// TIA Portal V17 export
// export: Created 2026-07-07T17:35:54.3389867Z, ExportSetting WithDefaults, DisplayName Totally Integrated Automation Portal, DisplayVersion V17, DisplayName TIA Portal Openness, DisplayVersion V17, DisplayName TIA Portal Version Control Interface, DisplayVersion V17, DisplayName STEP 7 Professional, DisplayVersion V17, DisplayName STEP 7 Safety, DisplayVersion V17, DisplayName WinCC Professional, DisplayVersion V17
FUNCTION_BLOCK "RS485_Com_Motor"   // FB2, LAD
TITLE = Feetech Motor with Cannet
{ S7_Optimized_Access := 'TRUE' }
VERSION : 0.1
// Note: Tcon block is required seperately for establishing the commincation.
// 
// Inputs:
// Connection_Done - Connection established bit from TCON block
// Slave_ID                  - Modbus RTU slave ID
// Target_Pos              - Input the Target position in Degrees
// Move                        - After giving the Target position this bit need to be enabled for executing. 
// 
// Outputs: 
// Actual_pos              - Gives the actual position in Degrees
// Target_Reached     - The bit will be enable for 2 seconds after the motor reaches the target position.
// stored: AutoNumber true, IsIECCheckEnabled false, IsRetainMemResEnabled false, MemoryReserve 100, SetENOAutomatically false, UDAEnableTagReadback false
   VAR_INPUT
      Connection_Done : Bool;
      Slave_ID : Int;
      Target_Pos : Int;
      Move : Bool;
   END_VAR
   VAR_OUTPUT
      "Actual_pos(Deg)" : Int;
      Target_Reached : Bool;
   END_VAR
   VAR
      CRC : Word;
      Frame_length : Int;
      CRC_Low : Byte;
      CRC_High : Byte;
      i : Int;
      j : Int;
      Data_Read { ExternalAccessible := 'False'; ExternalVisible := 'False'; ExternalWritable := 'False'} : Array[0..6] of Byte;
      Data_Write { ExternalAccessible := 'False'; ExternalVisible := 'False'; ExternalWritable := 'False'} : Array[0..7] of Byte;
      T_Send_block { S7_SetPoint := 'True'} : TSEND;
      T_RCV_Block { S7_SetPoint := 'True'} : TRCV;
      Move_timer { S7_SetPoint := 'True'} : IEC_TIMER;
      Send_req { S7_SetPoint := 'True'} : Bool;
      Function_code : Byte;
      Addr_low : Byte;
      Addr_high : Byte;
      Data_low : Byte;
      Data_high : Byte;
      Data_word : Word;
      Actual_pos_word : Word;
      Target_reach_timer : IEC_TIMER;
      Upper_limit { S7_SetPoint := 'True'} : Int;
      Lower_limit { S7_SetPoint := 'True'} : Int;
   END_VAR
BEGIN

REGION Network 1: Data send and recive
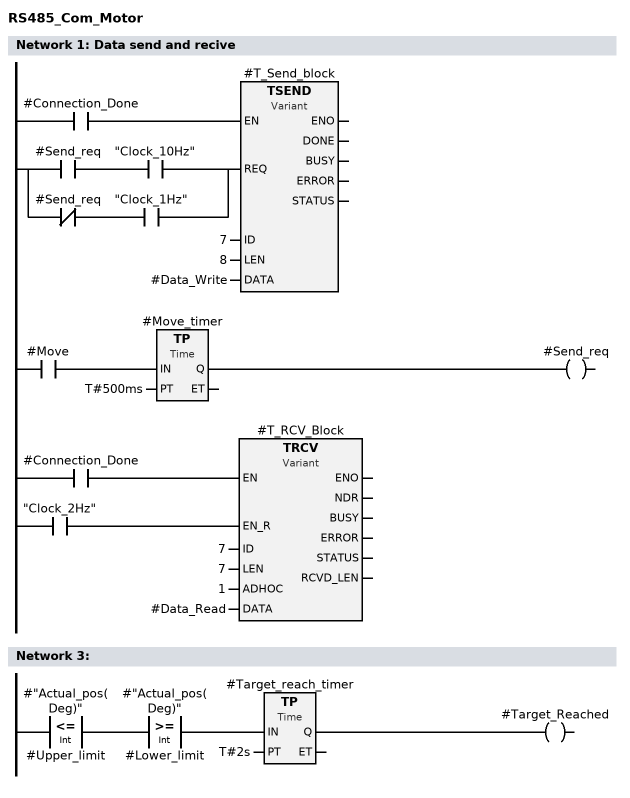
   RUNG wire#powerrail
      Contact( #Connection_Done )
      { S7_Templates := "[data_type := Variant, len_type := UDInt, id_type := CONN_OUC]" } #T_Send_block.TSEND(REQ := wire#w1, ID := 7, LEN := 8, DATA := #Data_Write, DONE =>, BUSY =>, ERROR =>, STATUS =>)
   END_RUNG
   RUNG wire#powerrail
      Contact( #Send_req )
      Contact( "Clock_10Hz" )
   END_RUNG wire#w1
   RUNG wire#powerrail
      I_Contact( #Send_req )
      Contact( "Clock_1Hz" )
   END_RUNG wire#w1
   RUNG wire#powerrail
      Contact( #Move )
      { S7_Templates := "time_type := Time" } #Move_timer.TP(pt := T#500ms, et =>)
      Coil( #Send_req )
   END_RUNG
   RUNG wire#powerrail
      Contact( #Connection_Done )
      { S7_Templates := "[card := 1, ptr_type := Variant, value_type := UDInt, id_type := CONN_OUC]" } #T_RCV_Block.TRCV(EN_R := wire#w2, ID := 7, LEN := 7, ADHOC := 1, DATA := #Data_Read, NDR =>, BUSY =>, ERROR =>, STATUS =>, RCVD_LEN =>)
   END_RUNG
   RUNG wire#powerrail
      Contact( "Clock_2Hz" )
   END_RUNG wire#w2
   // the same network as SCL:
   IF #Connection_Done THEN
       #T_Send_block(REQ := (#Send_req AND "Clock_10Hz") OR (NOT #Send_req AND "Clock_1Hz"),   // TSEND
                     ID := 7,
                     LEN := 8,
                     DATA := #Data_Write);
   END_IF;
   #Move_timer.TP(IN := #Move, PT := T#500ms);
   #Send_req := #Move_timer.Q;
   IF #Connection_Done THEN
       #T_RCV_Block(EN_R := "Clock_2Hz", ID := 7, LEN := 7, ADHOC := 1, DATA := #Data_Read);   // TRCV
   END_IF;
END_REGION

REGION Network 2 (SCL): Data move
   //Condition
   #Data_word := #Target_Pos * 10;

   IF #Send_req THEN
       #Function_code := 16#06;
       #Addr_low := 16#00;
       #Addr_high := 16#80;
       #Data_low := #Data_word.%B1;
       #Data_high := #Data_word.%B0;
   ELSE
       #Function_code := 16#03;
       #Addr_low := 16#01;
       #Addr_high := 16#01;
       #Data_low := 16#00;
       #Data_high := 16#01;
   END_IF;

   //Write Data

   #Data_Write[0] := #Slave_ID;
   #Data_Write[1] := #Function_code;
   #Data_Write[2] := #Addr_low;
   #Data_Write[3] := #Addr_high;
   #Data_Write[4] := #Data_low;
   #Data_Write[5] := #Data_high;
   #Data_Write[6] := #CRC_Low;
   #Data_Write[7] := #CRC_High;

   //Read Data

   IF #Data_Read[1] = 16#03 AND NOT #Send_req THEN
       #Actual_pos_word := #Data_Read[3];
       #Actual_pos_word := (SHL_WORD(IN := #Actual_pos_word, N := 8)) + #Data_Read[4];
       #"Actual_pos(Deg)" := WORD_TO_INT(#Actual_pos_word) / 10;

   END_IF;

   //Upper or lower limit definition

   #Upper_limit := #Target_Pos + 1;
   #Lower_limit := #Target_Pos - 1;
END_REGION

REGION Network 3
   RUNG wire#powerrail
      { S7_Templates := "SrcType := Int" } LE_Contact(in1 := #"Actual_pos(Deg)", in2 := #Upper_limit)
      { S7_Templates := "SrcType := Int" } GE_Contact(in1 := #"Actual_pos(Deg)", in2 := #Lower_limit)
      { S7_Templates := "time_type := Time" } #Target_reach_timer.TP(pt := T#2s, et =>)
      Coil( #Target_Reached )
   END_RUNG
   // the same network as SCL:
   #Target_reach_timer.TP(IN := (#"Actual_pos(Deg)" <= #Upper_limit) AND (#"Actual_pos(Deg)" >= #Lower_limit),
                          PT := T#2s);
   #Target_Reached := #Target_reach_timer.Q;
END_REGION

REGION Network 4 (SCL): CRC_Calculation
   #CRC := 16#FFFF;
   #Frame_length := 8;

   FOR #i := 0 TO #Frame_length - 3 DO

       #CRC := #CRC XOR #Data_Write[#i];

       FOR #j := 0 TO 7 DO

           IF (#CRC AND 1) = 1 THEN
               #CRC := SHR(IN := #CRC, N := 1);
               #CRC := #CRC XOR 16#A001;
           ELSE
               #CRC := SHR(IN := #CRC, N := 1);
           END_IF;

       END_FOR;

   END_FOR;
   #CRC_Low := WORD_TO_BYTE(#CRC AND 16#00FF);
   #CRC_High := WORD_TO_BYTE(SHR(IN:=#CRC, N:=8));
END_REGION
END_FUNCTION_BLOCK
